{attribute 'no_explicit_call':= 'do not call this POU directly'}
FUNCTION_BLOCK T_ValueMonitorEx
VAR
    _Changed    : BOOL;
    StoredValue : ARRAY[0..7] OF BYTE;
END_VAR

PROPERTY Changed : BOOL
GET
Changed := _Changed;
END_GET
END_PROPERTY

METHOD Reset
VAR_INPUT
END_VAR
MEMSET(destAddr := ADR(StoredValue),
       fillByte := 16#00,
       n        := SIZEOF(StoredValue));
END_METHOD

METHOD Test : BOOL;
VAR_INPUT
    Value : ANY_NUM;
END_VAR
_Changed := 0 <>
            MEMCMP(pBuf1 := Value.pValue,
                   pBuf2 := ADR(StoredValue),
                   n     := DINT_TO_UDINT(Value.diSize));

IF _Changed THEN
    MEMCPY(destAddr := ADR(StoredValue),
           srcAddr  := Value.pValue,
           n        := DINT_TO_UDINT(Value.diSize));
END_IF

Test := _Changed;
END_METHOD

END_FUNCTION_BLOCK

(* stored: Version 1.1.0.1, ProductVersion 3.1.4024.12
   POU T_ValueMonitorEx: Id {bacae591-70bd-03f3-1d52-321cbceb26da}, SpecialFunc None
   Property Changed: Id {51edbcfe-dede-04c7-0459-a6015be2ca88}
   Get Get: Id {99977f8b-4a89-07a7-3d53-1ff3084f751a}
   Method Reset: Id {0b7c1ee6-a5c4-0d75-1e2b-580f2737e28e}
   Method Test: Id {24bc92f7-bd36-0ba0-0222-49588d079fd0} *)
